VAR
    bStatus : BOOL := FALSE; // or TRUE
END_VAR

(* stored: Version 1.1.0.1, ProductVersion 3.1.4024.13
   POU MAIN: Id {bb009617-2d4f-4999-a2b9-f4b71b49f1b6}, SpecialFunc None *)
